// TIA Portal V17 export
// export: Created 2025-06-25T13:13:28.2176113Z, ExportSetting WithDefaults, DisplayName Totally Integrated Automation Portal, DisplayVersion V17 Update 8, DisplayName TIA Portal Openness, DisplayVersion V17 Update 8, DisplayName TIA Portal Version Control Interface, DisplayVersion V17, DisplayName STEP 7 Professional, DisplayVersion V17 Update 8, DisplayName STEP 7 Safety, DisplayVersion V17 Update 6, DisplayName WinCC Advanced, DisplayVersion V17 Update 8
TYPE "stET200AL_DIQ_Q"
// stored: IsFailsafeCompliant false
   STRUCT
      DQ00 : Bool;
      DQ01 : Bool;
      DQ02 : Bool;
      DQ03 : Bool;
      DQ04 : Bool;
      DQ05 : Bool;
      DQ06 : Bool;
      DQ07 : Bool;
      DQ08 : Bool;
      DQ09 : Bool;
      DQ10 : Bool;
      DQ11 : Bool;
      DQ12 : Bool;
      DQ13 : Bool;
      DQ14 : Bool;
      DQ15 : Bool;
   END_STRUCT;
END_TYPE
